// TIA Portal V19 export
// export: Created 2026-08-09T01:52:25.7899977Z, ExportSetting WithDefaults, DisplayName Totally Integrated Automation Portal, DisplayVersion V19, DisplayName TIA Portal Openness, DisplayVersion V19, DisplayName TIA Portal Version Control Interface, DisplayVersion V19, DisplayName STEP 7 Professional, DisplayVersion V19, DisplayName STEP 7 Safety, DisplayVersion V19, DisplayName WinCC Basic/Comfort/Advanced, DisplayVersion V19, DisplayName WinCC Unified, DisplayVersion V19
FUNCTION_BLOCK "dc"   // FB1, LAD
{ S7_Optimized_Access := 'TRUE' }
VERSION : 0.1
// stored: AutoNumber true, IsIECCheckEnabled false, IsRetainMemResEnabled false, MemoryReserve 100, SetENOAutomatically false, UDAEnableTagReadback false
   VAR_INPUT
      timePt : Time;
   END_VAR
   VAR_OUTPUT
      timeQ : Bool;
   END_VAR
   VAR
      timeP : Bool;
      timeS : Bool;
   END_VAR
BEGIN

REGION Network 1
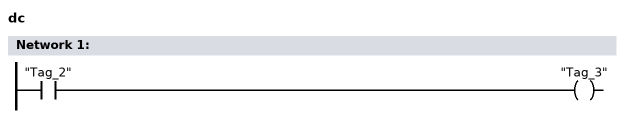
   RUNG wire#powerrail
      Contact( "Tag_2" )
      Coil( "Tag_3" )
   END_RUNG
   // the same network as SCL:
   "Tag_3" := "Tag_2";
END_REGION

REGION Network 3 (SCL)
   "IEC_Timer_0_DB".TON(IN:=#timeS,
                        PT:=#timePt,
                        Q=>#timeQ);

   IF "Tag_4" THEN
       "Tag_5" := TRUE;
       #timeS := FALSE;
   ELSE
       "Tag_5" := FALSE;
       #timeS := TRUE;
   END_IF;
END_REGION
END_FUNCTION_BLOCK
